// TIA Portal V19 export
ORGANIZATION_BLOCK "Startup"   // OB2000, LAD, Startup
TITLE = "Complete Restart"
// This block is called only once in the very first PLC cycle after STOP -> RUN.
// Configuration seetings and assignemts are to be programmed here.
// stored: AutoNumber false, IsIECCheckEnabled true, Namespace Unit, SetENOAutomatically true
   VAR_INPUT
      LostRetentive : Bool;   // True if retentive data are lost
      LostRTC : Bool;   // True if date and time are lost
   END_VAR
BEGIN

REGION Network 1 (SCL): Build the Absolut Reference Designator
   // Set the Absoult Reference Designator in the DB Config. It is combined out of the parent reference designator and the own reference designator (=relative)
   IF LEN(IN := "Unit.Config".unit.referenceDesignator.parent) <> 0 THEN
       "Unit.Config".unit.referenceDesignator.combined := CONCAT_WSTRING(IN1 := "Unit.Config".unit.referenceDesignator.parent, IN2 := WSTRING#'.', IN3 := "Unit.Config".unit.referenceDesignator.relative);
   ELSE
       "Unit.Config".unit.referenceDesignator.combined := "Unit.Config".unit.referenceDesignator.relative;
   END_IF;
END_REGION

REGION Network 2: Configuration of the OMAC State Machine
   // In the DB Config, the state machine can be configured in a convenient way. LUC_StateMachineConfig translates that configuration into the configuration variables for the stateModeManager.
   // Additionally, the EnabledModes are copied to the interface so that they can be shown on the HMI.
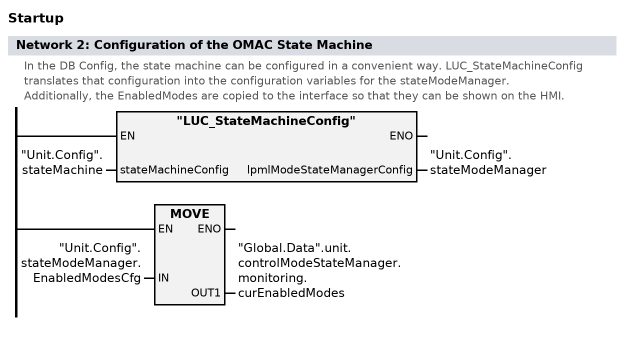
   RUNG wire#powerrail
      "LUC_StateMachineConfig"(stateMachineConfig := "Unit.Config".stateMachine, lpmlModeStateManagerConfig => "Unit.Config".stateModeManager)
   END_RUNG
   RUNG wire#powerrail
      Move(in := "Unit.Config".stateModeManager.EnabledModesCfg, out1 => "Global.Data".unit.controlModeStateManager.monitoring.curEnabledModes)
   END_RUNG
   // the same network as SCL:
   "LUC_StateMachineConfig"(stateMachineConfig := "Unit.Config".stateMachine,
                           lpmlModeStateManagerConfig => "Unit.Config".stateModeManager);
   "Global.Data".unit.controlModeStateManager.monitoring.curEnabledModes := "Unit.Config".stateModeManager.EnabledModesCfg;
END_REGION
END_ORGANIZATION_BLOCK
